(* CODESYS project Timestamp.gvl.xml

Project tree, tasks and I/O mapping:
  global variables Timestamp
*)

// Timestamp
{attribute 'qualified_only'}
VAR_GLOBAL
	Current: SysTime;
	UTC: SysTimeDate;
	Local: SysTimeDate;
END_VAR
